// TIA Portal V18 export
DATA_BLOCK "AndonMain_DB"   // DB5
VERSION : 0.1
// stored: AutoNumber true, DBAccessibleFromOPCUA true, DBAccessibleFromWebserver true, InstanceOfName AndonMain, InstanceOfType FB
"AndonMain"
   // VAR
   //    fpBit_greenTrigger : Bool;
   //    AndonBoxASi_v2_Instance_8 { S7_SetPoint := 'True'} : "AndonBoxASi";
   //    AndonBoxASi_v2_Instance_9 { S7_SetPoint := 'True'} : "AndonBoxASi";
   //    AndonBoxASi_v2_Instance1 { S7_SetPoint := 'True'} : "AndonBoxASi";
   //    AndonBoxASi_v2_Instance2 { S7_SetPoint := 'True'} : "AndonBoxASi";
   //    AndonBoxASi_v2_Instance3 { S7_SetPoint := 'True'} : "AndonBoxASi";
   //    AndonBoxASi_v2_Instance4 { S7_SetPoint := 'True'} : "AndonBoxASi";
   //    AndonBoxASi_v2_Instance5 { S7_SetPoint := 'True'} : "AndonBoxASi";
   //    AndonBoxASi_v2_Instance6 { S7_SetPoint := 'True'} : "AndonBoxASi";
   //    AndonBoxASi_v2_Instance7 { S7_SetPoint := 'True'} : "AndonBoxASi";
   //    AndonBoxASi_v2_Instance10 { S7_SetPoint := 'True'} : "AndonBoxASi";
   // END_VAR
BEGIN
END_DATA_BLOCK
